(* Logix 5000 project; controller cal1632 1756-L62 rev 16.20; software revision 16.05; part 19 of 61 *)
(* tags used below, declared in another part *)
   FAULT : BOOL;
   p01_param_fan_zero_speed : REAL;
   p01_param_open_oven_recirc_sp : REAL;
   p01_param_temp_limit : REAL;
   p01_recipe_active : recipe;
   p01r02 : routine;
   p01r09_open_oven : BOOL;
   p01r09_pb_global_reset : BOOL;
   p02_dint_from_hmi : hmi_dint;
   p11r02_shutdown_temp : BOOL;
   p11r30 : routine;
   p12_ai_recirc_rpm : REAL;
   p12_ao_recirc_selected_speed : REAL;
   p12_di_recirc : acs800_di_normal;
   p12_di_recirc_fan_mtr_ts : BOOL;
   p12_di_recirc_flow_ok : BOOL;
   p12_do_recirc : acs800_do_normal;
   p12r02_shutdown_temp : BOOL;
   p12r20_state : DINT;
   p12r30 : routine;
   p12r32 : routine;
   p12r32_fan_pb_stopped : BOOL;
   p12r32_pb_start : BOOL;
   p12r32_pb_stop : BOOL;
   p12r32_request_auto_run : BOOL;
   p12r32_run_permissive : BOOL;
   p12r32_timer_fault : TIMER[5];
   p12r32_timer_warning : TIMER[5];
   p12r32_vfd_stopped : BOOL;
   p13_ai_exhaust_amps : REAL;
   p13_ai_exhaust_hz : REAL;
   p13_ai_exhaust_hz_max : REAL;
   p13_ai_exhaust_rpm : REAL;
   p13_ai_recirc_amps : REAL;
   p13_ai_recirc_hz : REAL;
   p13_ai_recirc_hz_max : REAL;
   p13_ai_recirc_rpm : REAL;
   p13_ai_tc01 : REAL;
   p13_ai_tc02 : REAL;
   p13_di_door_open : BOOL;
   p13_di_exh : acs800_di_normal;
   p13_di_exh_fan_mtr_ts : BOOL;
   p13_di_exh_flow_ok : BOOL;
   p13_di_filter_clean : BOOL;
   p13_di_recirc : acs800_di_normal;
   p13_di_recirc_fan_mtr_ts : BOOL;
   p13_di_recirc_flow_ok : BOOL;
   p13_di_tc01_bo : BOOL;
   p13_di_tc02_bo : BOOL;
   p13_dint_to_hmi : DINT[16];
   p13_param_shutdown_temp : REAL;
   p13_param_tc01z : REAL;
   p13_param_tc02z : REAL;
   p13r01 : routine;
   p13r02 : routine;
   p13r02_fault_exists : BOOL;
   p13r02_not_safe_temp : BOOL;
   p13r02_safe_temp : BOOL;
   p13r02_shutdown_temp : BOOL;
   p13r02_timer_fault : TIMER[4];
   p13r02_timer_safe_temp : TIMER[2];
   p13r02_timer_warning : TIMER[4];
   p13r02_unack_fault : BOOL;
   p13r02_unack_warning : BOOL;
   p13r02_warning_exists : BOOL;
   p13r03 : routine;
   p13r03_hz : SYS_SCP;
   p13r03_timer_fault : TIMER[4];
   p13r03_timer_warning : TIMER[4];
   p13r04 : routine;
   p13r05 : routine;
   p13r06 : routine;
   p13r07 : routine;
   p13r08 : routine;
   p13r09 : routine;
   p13r10 : routine;
   p13r20 : routine;
   p13r30 : routine;
   p13r31 : routine;
   p13r32 : routine;
   p23r02 : routine;
(* P12_Zone_2, continued *)

ROUTINE R32_Recirc_VFD   (* ladder *)
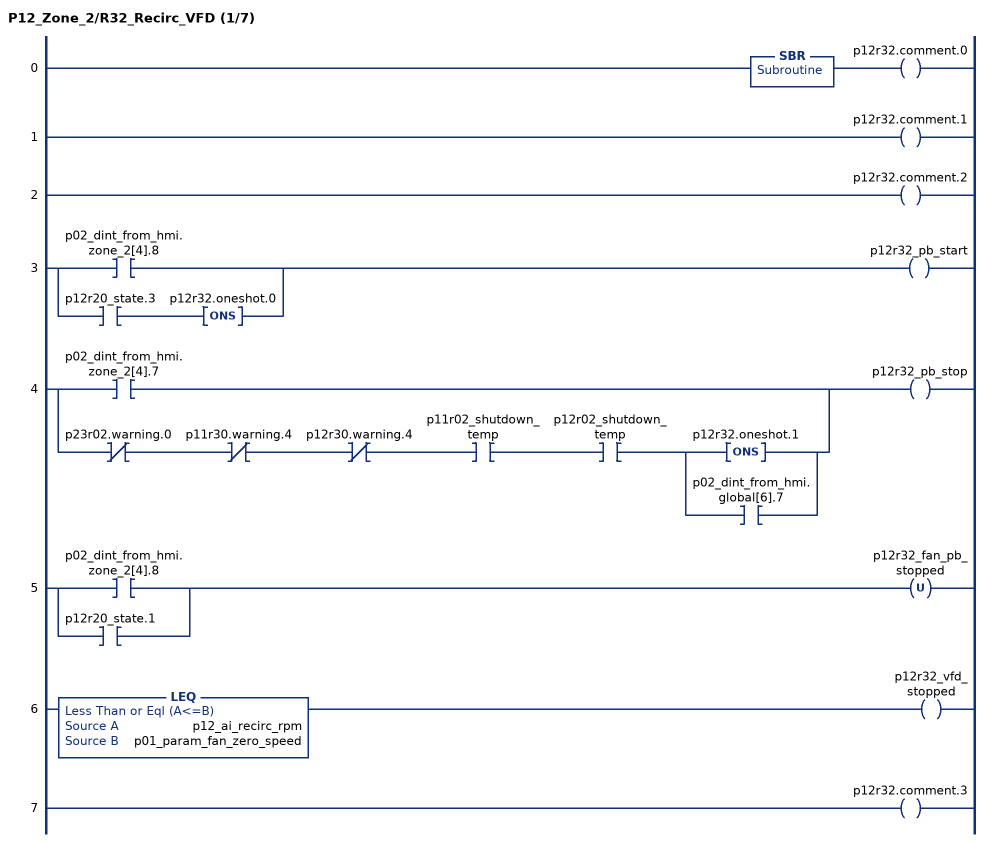
   0: SBR()OTE(p12r32.comment.0);
   1: OTE(p12r32.comment.1);
   2: OTE(p12r32.comment.2);
   3: [XIC(p02_dint_from_hmi.zone_2[4].8) ,XIC(p12r20_state.3) ONS(p12r32.oneshot.0) ]OTE(p12r32_pb_start);
   4: [XIC(p02_dint_from_hmi.zone_2[4].7) ,XIO(p23r02.warning.0) XIO(p11r30.warning.4) XIO(p12r30.warning.4) XIC(p11r02_shutdown_temp) XIC(p12r02_shutdown_temp) [ONS(p12r32.oneshot.1) ,XIC(p02_dint_from_hmi.global[6].7) ] ]OTE(p12r32_pb_stop);
   5: [XIC(p02_dint_from_hmi.zone_2[4].8) ,XIC(p12r20_state.1) ]OTU(p12r32_fan_pb_stopped);
   6: LEQ(p12_ai_recirc_rpm,p01_param_fan_zero_speed)OTE(p12r32_vfd_stopped);
   7: OTE(p12r32.comment.3);
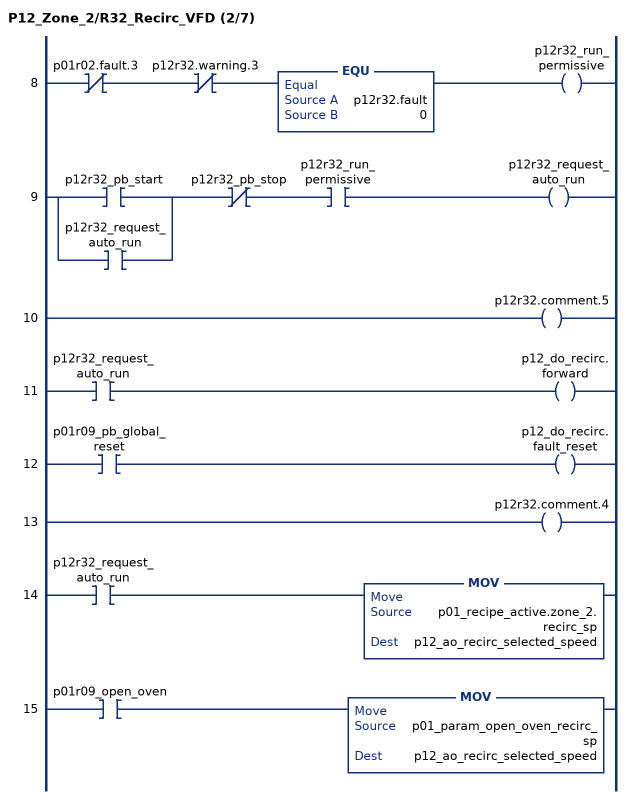
   8: XIO(p01r02.fault.3)XIO(p12r32.warning.3)EQU(p12r32.fault,0)OTE(p12r32_run_permissive);
   9: [XIC(p12r32_pb_start) ,XIC(p12r32_request_auto_run) ]XIO(p12r32_pb_stop)XIC(p12r32_run_permissive)OTE(p12r32_request_auto_run);
   10: OTE(p12r32.comment.5);
   11: XIC(p12r32_request_auto_run)OTE(p12_do_recirc.forward);
   12: XIC(p01r09_pb_global_reset)OTE(p12_do_recirc.fault_reset);
   13: OTE(p12r32.comment.4);
   14: XIC(p12r32_request_auto_run)MOV(p01_recipe_active.zone_2.recirc_sp,p12_ao_recirc_selected_speed);
   15: XIC(p01r09_open_oven)MOV(p01_param_open_oven_recirc_sp,p12_ao_recirc_selected_speed);
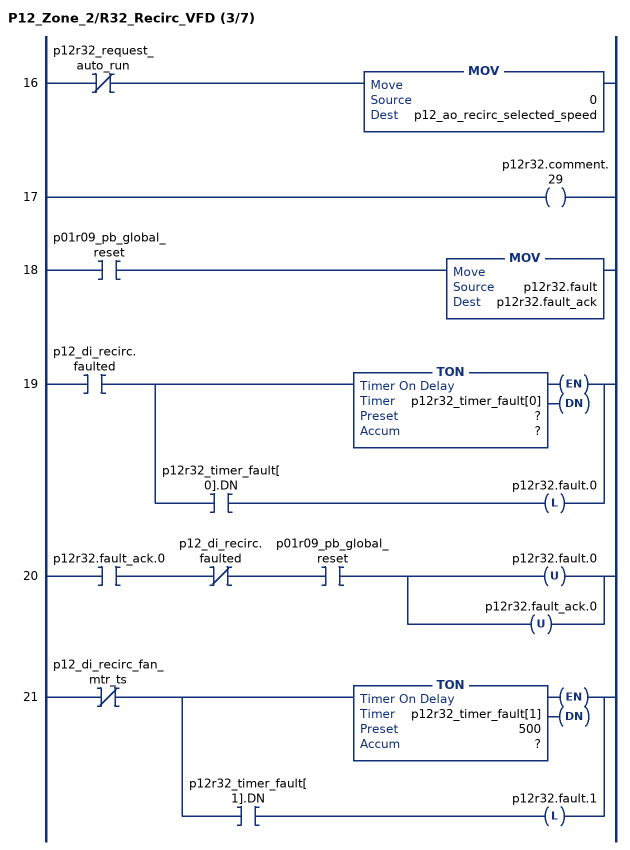
   16: XIO(p12r32_request_auto_run)MOV(0,p12_ao_recirc_selected_speed);
   17: OTE(p12r32.comment.29);
   18: XIC(p01r09_pb_global_reset)MOV(p12r32.fault,p12r32.fault_ack);
   19: XIC(p12_di_recirc.faulted)[TON(p12r32_timer_fault[0],?,?) ,XIC(p12r32_timer_fault[0].DN) OTL(p12r32.fault.0) ];
   20: XIC(p12r32.fault_ack.0)XIO(p12_di_recirc.faulted)XIC(p01r09_pb_global_reset)[OTU(p12r32.fault.0) ,OTU(p12r32.fault_ack.0) ];
   21: XIO(p12_di_recirc_fan_mtr_ts)[TON(p12r32_timer_fault[1],?,?) ,XIC(p12r32_timer_fault[1].DN) OTL(p12r32.fault.1) ];
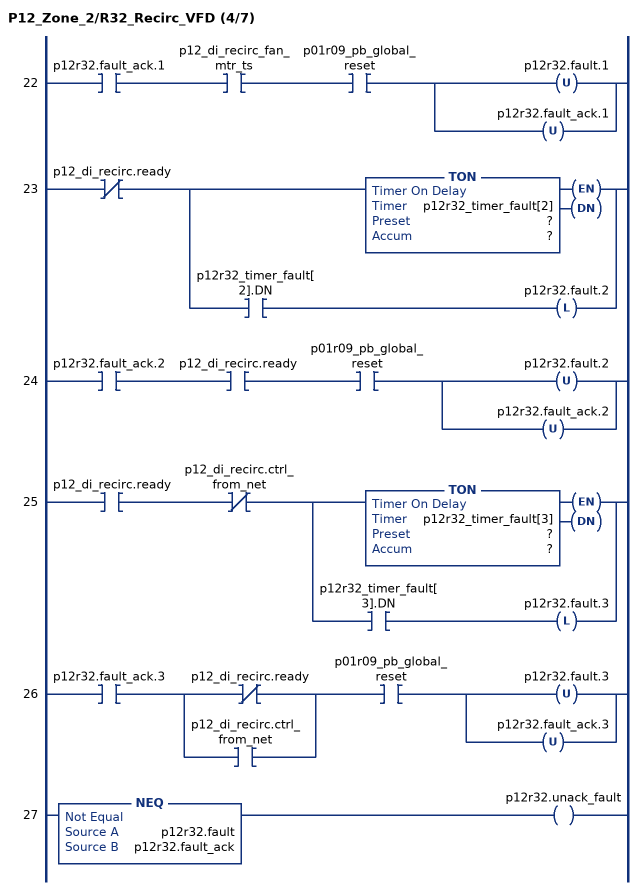
   22: XIC(p12r32.fault_ack.1)XIC(p12_di_recirc_fan_mtr_ts)XIC(p01r09_pb_global_reset)[OTU(p12r32.fault.1) ,OTU(p12r32.fault_ack.1) ];
   23: XIO(p12_di_recirc.ready)[TON(p12r32_timer_fault[2],?,?) ,XIC(p12r32_timer_fault[2].DN) OTL(p12r32.fault.2) ];
   24: XIC(p12r32.fault_ack.2)XIC(p12_di_recirc.ready)XIC(p01r09_pb_global_reset)[OTU(p12r32.fault.2) ,OTU(p12r32.fault_ack.2) ];
   25: XIC(p12_di_recirc.ready)XIO(p12_di_recirc.ctrl_from_net)[TON(p12r32_timer_fault[3],?,?) ,XIC(p12r32_timer_fault[3].DN) OTL(p12r32.fault.3) ];
   26: XIC(p12r32.fault_ack.3)[XIO(p12_di_recirc.ready) ,XIC(p12_di_recirc.ctrl_from_net) ]XIC(p01r09_pb_global_reset)[OTU(p12r32.fault.3) ,OTU(p12r32.fault_ack.3) ];
   27: NEQ(p12r32.fault,p12r32.fault_ack)OTE(p12r32.unack_fault);
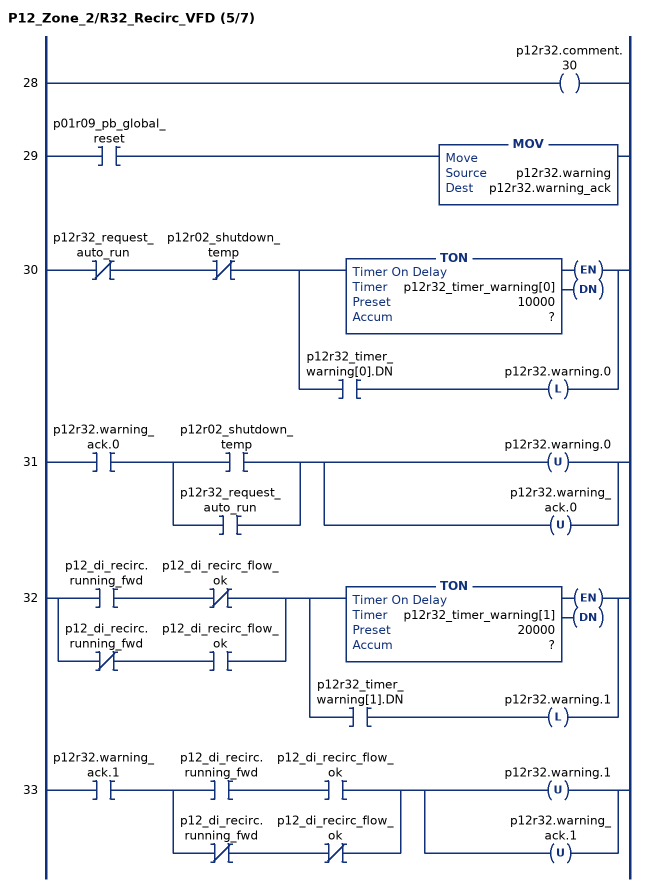
   28: OTE(p12r32.comment.30);
   29: XIC(p01r09_pb_global_reset)MOV(p12r32.warning,p12r32.warning_ack);
   30: XIO(p12r32_request_auto_run)XIO(p12r02_shutdown_temp)[TON(p12r32_timer_warning[0],?,?) ,XIC(p12r32_timer_warning[0].DN) OTL(p12r32.warning.0) ];
   31: XIC(p12r32.warning_ack.0)[XIC(p12r02_shutdown_temp) ,XIC(p12r32_request_auto_run) ][OTU(p12r32.warning.0) ,OTU(p12r32.warning_ack.0) ];
   32: [XIC(p12_di_recirc.running_fwd) XIO(p12_di_recirc_flow_ok) ,XIO(p12_di_recirc.running_fwd) XIC(p12_di_recirc_flow_ok) ][TON(p12r32_timer_warning[1],?,?) ,XIC(p12r32_timer_warning[1].DN) OTL(p12r32.warning.1) ];
   33: XIC(p12r32.warning_ack.1)[XIC(p12_di_recirc.running_fwd) XIC(p12_di_recirc_flow_ok) ,XIO(p12_di_recirc.running_fwd) XIO(p12_di_recirc_flow_ok) ][OTU(p12r32.warning.1) ,OTU(p12r32.warning_ack.1) ];
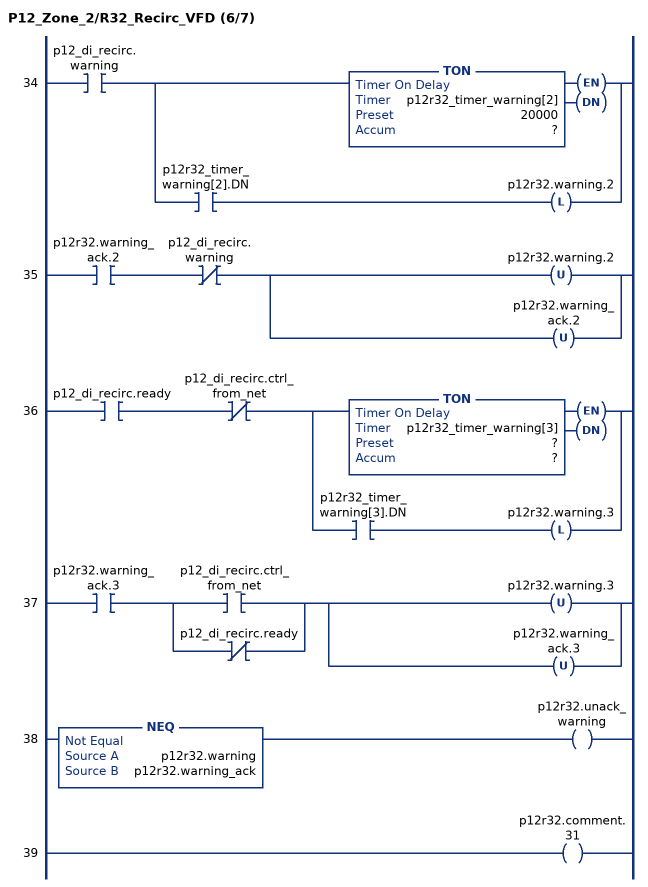
   34: XIC(p12_di_recirc.warning)[TON(p12r32_timer_warning[2],?,?) ,XIC(p12r32_timer_warning[2].DN) OTL(p12r32.warning.2) ];
   35: XIC(p12r32.warning_ack.2)XIO(p12_di_recirc.warning)[OTU(p12r32.warning.2) ,OTU(p12r32.warning_ack.2) ];
   36: XIC(p12_di_recirc.ready)XIO(p12_di_recirc.ctrl_from_net)[TON(p12r32_timer_warning[3],?,?) ,XIC(p12r32_timer_warning[3].DN) OTL(p12r32.warning.3) ];
   37: XIC(p12r32.warning_ack.3)[XIC(p12_di_recirc.ctrl_from_net) ,XIO(p12_di_recirc.ready) ][OTU(p12r32.warning.3) ,OTU(p12r32.warning_ack.3) ];
   38: NEQ(p12r32.warning,p12r32.warning_ack)OTE(p12r32.unack_warning);
   39: OTE(p12r32.comment.31);
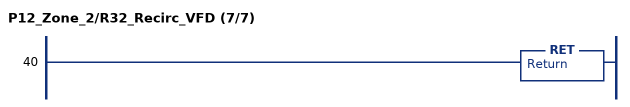
   40: RET();
END_ROUTINE
END_PROGRAM

PROGRAM P13_Zone_3   (* main routine R01_Main *)

ROUTINE R01_Main   (* ladder *)
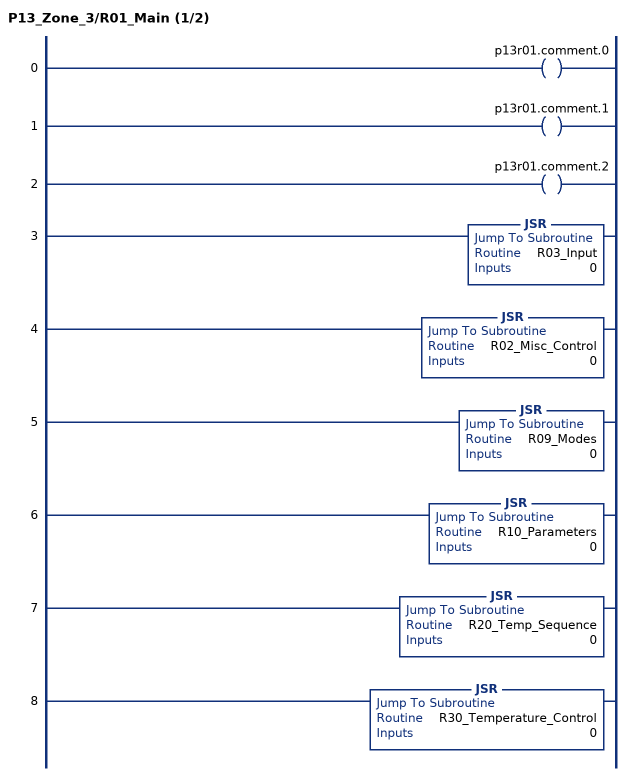
   0: OTE(p13r01.comment.0);
   1: OTE(p13r01.comment.1);
   2: OTE(p13r01.comment.2);
   3: JSR(R03_Input,0);
   4: JSR(R02_Misc_Control,0);
   5: JSR(R09_Modes,0);
   6: JSR(R10_Parameters,0);
   7: JSR(R20_Temp_Sequence,0);
   8: JSR(R30_Temperature_Control,0);
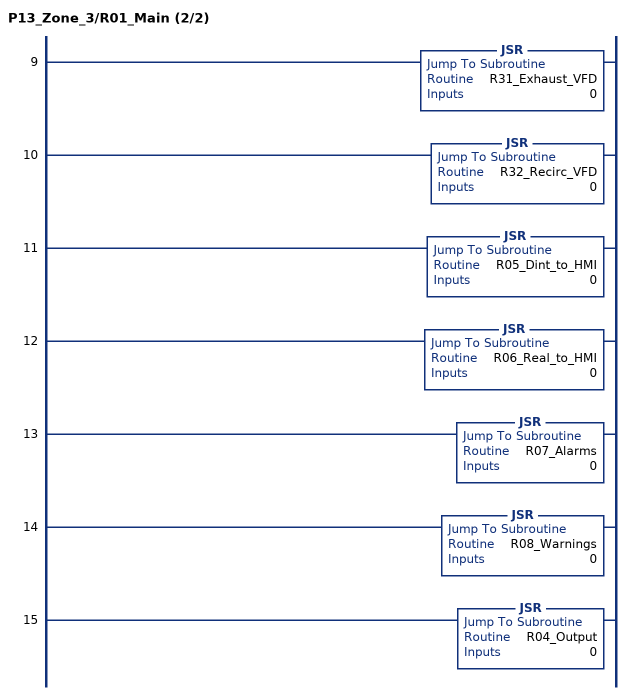
   9: JSR(R31_Exhaust_VFD,0);
   10: JSR(R32_Recirc_VFD,0);
   11: JSR(R05_Dint_to_HMI,0);
   12: JSR(R06_Real_to_HMI,0);
   13: JSR(R07_Alarms,0);
   14: JSR(R08_Warnings,0);
   15: JSR(R04_Output,0);
END_ROUTINE

ROUTINE R02_Misc_Control   (* ladder *)
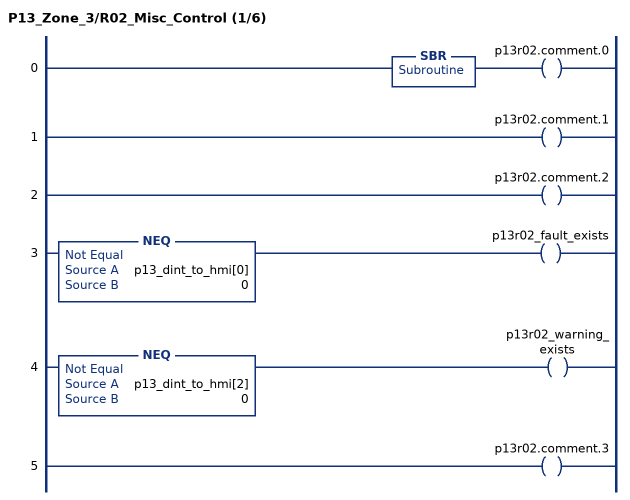
   0: SBR()OTE(p13r02.comment.0);
   1: OTE(p13r02.comment.1);
   2: OTE(p13r02.comment.2);
   3: NEQ(p13_dint_to_hmi[0],0)OTE(p13r02_fault_exists);
   4: NEQ(p13_dint_to_hmi[2],0)OTE(p13r02_warning_exists);
   5: OTE(p13r02.comment.3);
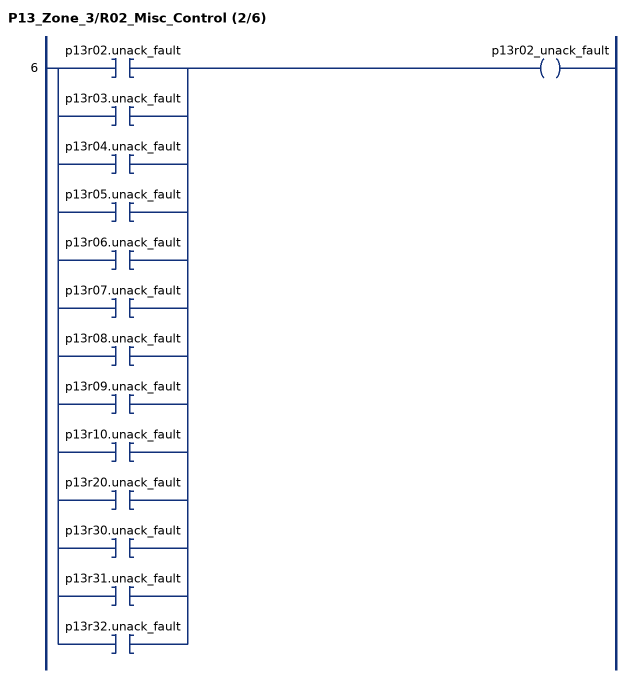
   6: [XIC(p13r02.unack_fault) ,XIC(p13r03.unack_fault) ,XIC(p13r04.unack_fault) ,XIC(p13r05.unack_fault) ,XIC(p13r06.unack_fault) ,XIC(p13r07.unack_fault) ,XIC(p13r08.unack_fault) ,XIC(p13r09.unack_fault) ,XIC(p13r10.unack_fault) ,XIC(p13r20.unack_fault) ,XIC(p13r30.unack_fault) ,XIC(p13r31.unack_fault) ,XIC(p13r32.unack_fault) ]OTE(p13r02_unack_fault);
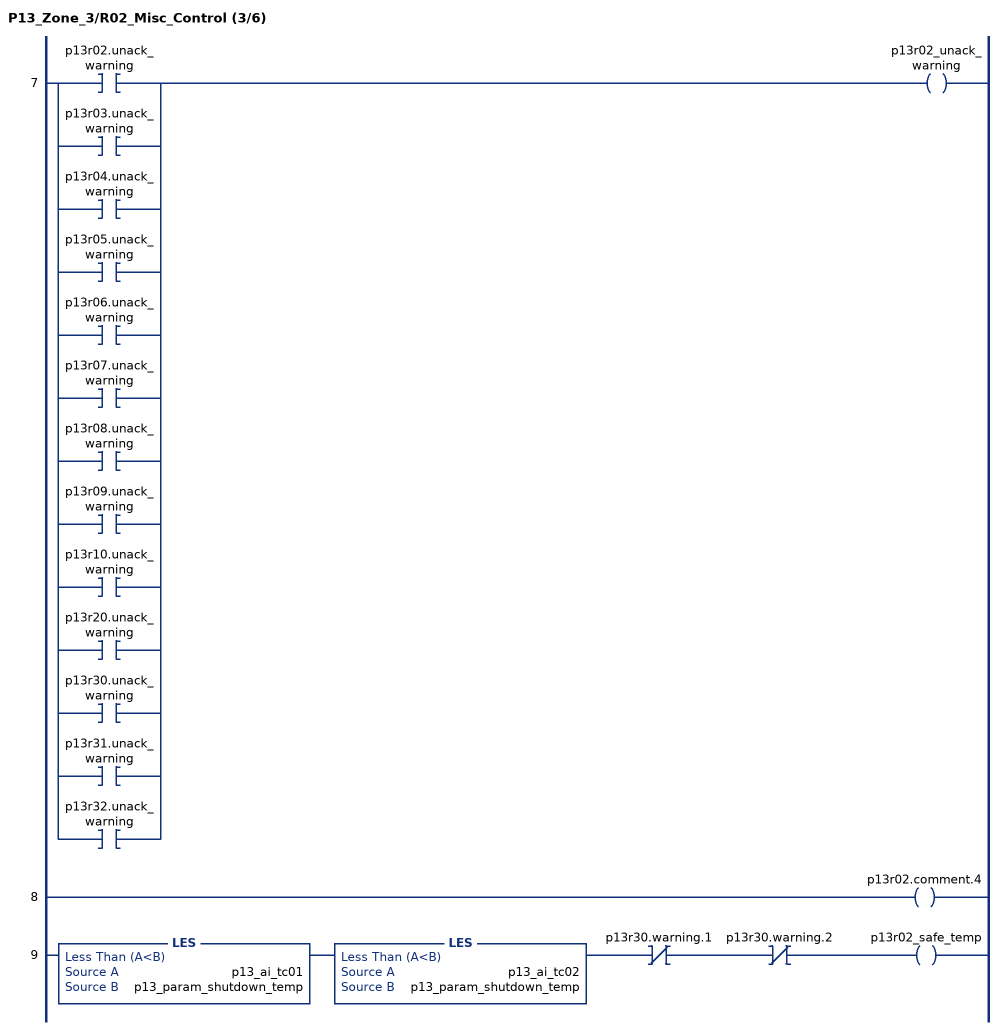
   7: [XIC(p13r02.unack_warning) ,XIC(p13r03.unack_warning) ,XIC(p13r04.unack_warning) ,XIC(p13r05.unack_warning) ,XIC(p13r06.unack_warning) ,XIC(p13r07.unack_warning) ,XIC(p13r08.unack_warning) ,XIC(p13r09.unack_warning) ,XIC(p13r10.unack_warning) ,XIC(p13r20.unack_warning) ,XIC(p13r30.unack_warning) ,XIC(p13r31.unack_warning) ,XIC(p13r32.unack_warning) ]OTE(p13r02_unack_warning);
   8: OTE(p13r02.comment.4);
   9: LES(p13_ai_tc01,p13_param_shutdown_temp)LES(p13_ai_tc02,p13_param_shutdown_temp)XIO(p13r30.warning.1)XIO(p13r30.warning.2)OTE(p13r02_safe_temp);
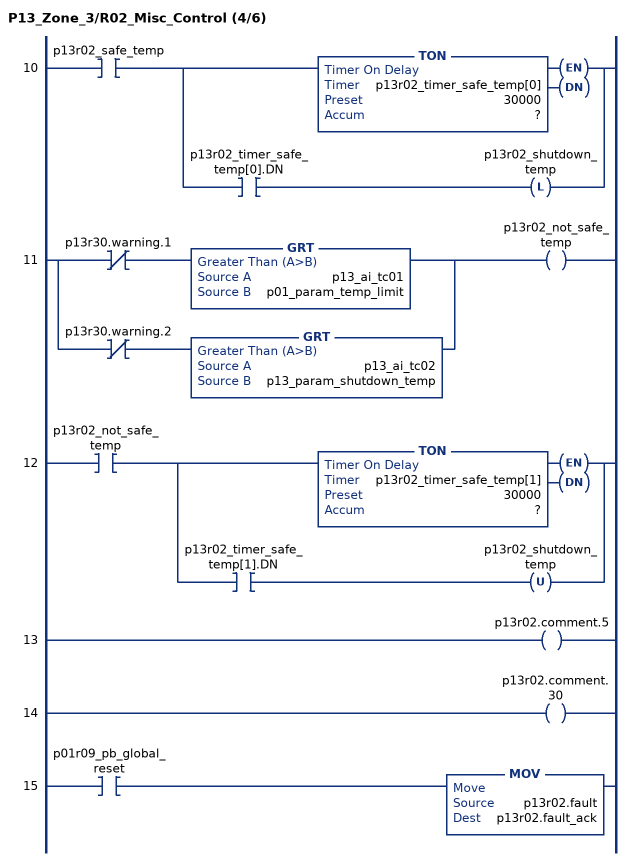
   10: XIC(p13r02_safe_temp)[TON(p13r02_timer_safe_temp[0],?,?) ,XIC(p13r02_timer_safe_temp[0].DN) OTL(p13r02_shutdown_temp) ];
   11: [XIO(p13r30.warning.1) GRT(p13_ai_tc01,p01_param_temp_limit) ,XIO(p13r30.warning.2) GRT(p13_ai_tc02,p13_param_shutdown_temp) ]OTE(p13r02_not_safe_temp);
   12: XIC(p13r02_not_safe_temp)[TON(p13r02_timer_safe_temp[1],?,?) ,XIC(p13r02_timer_safe_temp[1].DN) OTU(p13r02_shutdown_temp) ];
   13: OTE(p13r02.comment.5);
   14: OTE(p13r02.comment.30);
   15: XIC(p01r09_pb_global_reset)MOV(p13r02.fault,p13r02.fault_ack);
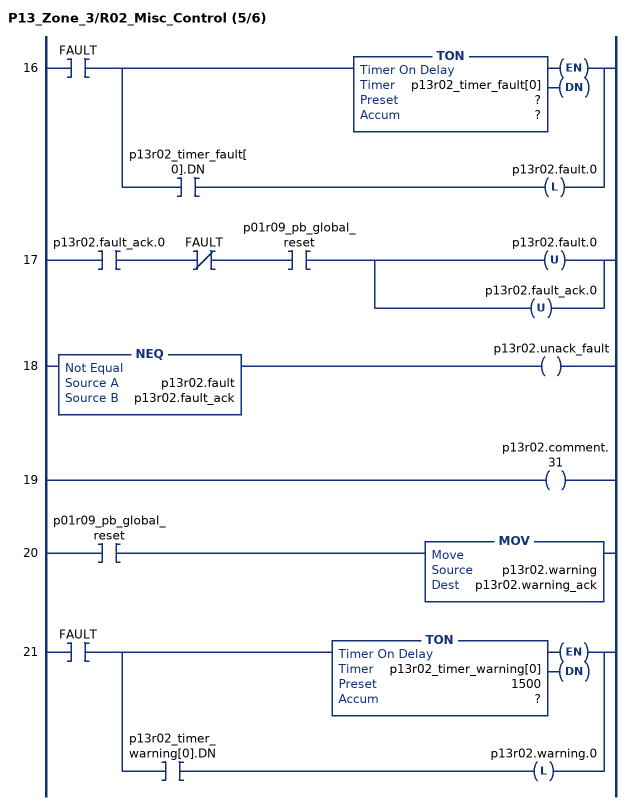
   16: XIC(FAULT)[TON(p13r02_timer_fault[0],?,?) ,XIC(p13r02_timer_fault[0].DN) OTL(p13r02.fault.0) ];
   17: XIC(p13r02.fault_ack.0)XIO(FAULT)XIC(p01r09_pb_global_reset)[OTU(p13r02.fault.0) ,OTU(p13r02.fault_ack.0) ];
   18: NEQ(p13r02.fault,p13r02.fault_ack)OTE(p13r02.unack_fault);
   19: OTE(p13r02.comment.31);
   20: XIC(p01r09_pb_global_reset)MOV(p13r02.warning,p13r02.warning_ack);
   21: XIC(FAULT)[TON(p13r02_timer_warning[0],?,?) ,XIC(p13r02_timer_warning[0].DN) OTL(p13r02.warning.0) ];
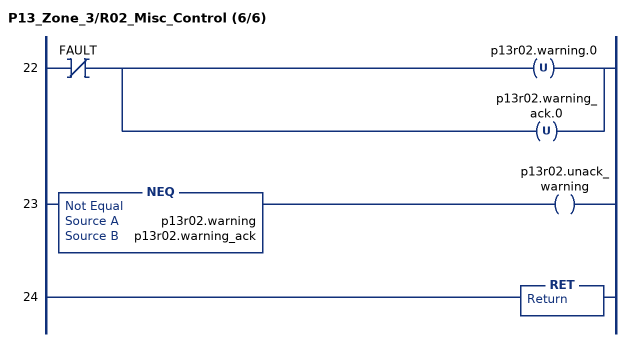
   22: XIO(FAULT)[OTU(p13r02.warning.0) ,OTU(p13r02.warning_ack.0) ];
   23: NEQ(p13r02.warning,p13r02.warning_ack)OTE(p13r02.unack_warning);
   24: RET();
END_ROUTINE

ROUTINE R03_Input   (* ladder *)
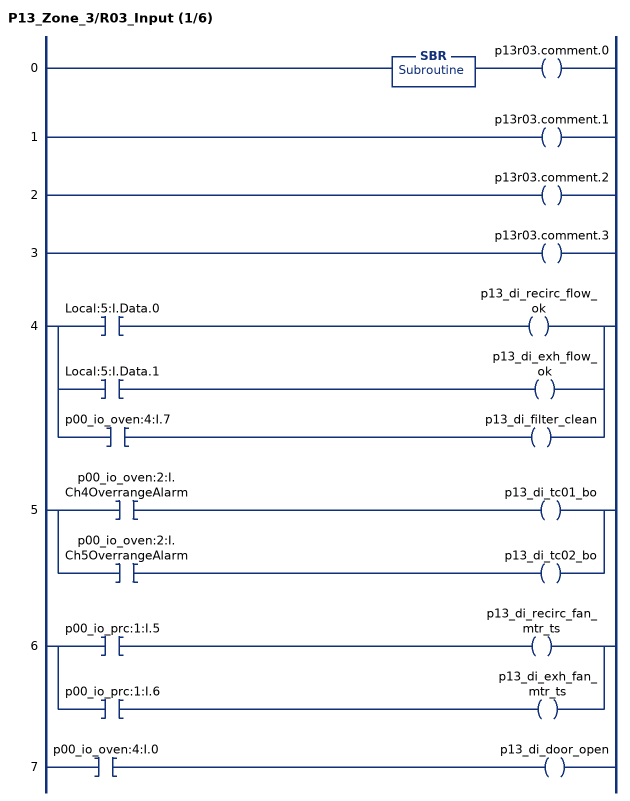
   0: SBR()OTE(p13r03.comment.0);
   1: OTE(p13r03.comment.1);
   2: OTE(p13r03.comment.2);
   3: OTE(p13r03.comment.3);
   4: [XIC(Local:5:I.Data.0) OTE(p13_di_recirc_flow_ok) ,XIC(Local:5:I.Data.1) OTE(p13_di_exh_flow_ok) ,XIC(p00_io_oven:4:I.7) OTE(p13_di_filter_clean) ];
   5: [XIC(p00_io_oven:2:I.Ch4OverrangeAlarm) OTE(p13_di_tc01_bo) ,XIC(p00_io_oven:2:I.Ch5OverrangeAlarm) OTE(p13_di_tc02_bo) ];
   6: [XIC(p00_io_prc:1:I.5) OTE(p13_di_recirc_fan_mtr_ts) ,XIC(p00_io_prc:1:I.6) OTE(p13_di_exh_fan_mtr_ts) ];
   7: XIC(p00_io_oven:4:I.0)OTE(p13_di_door_open);
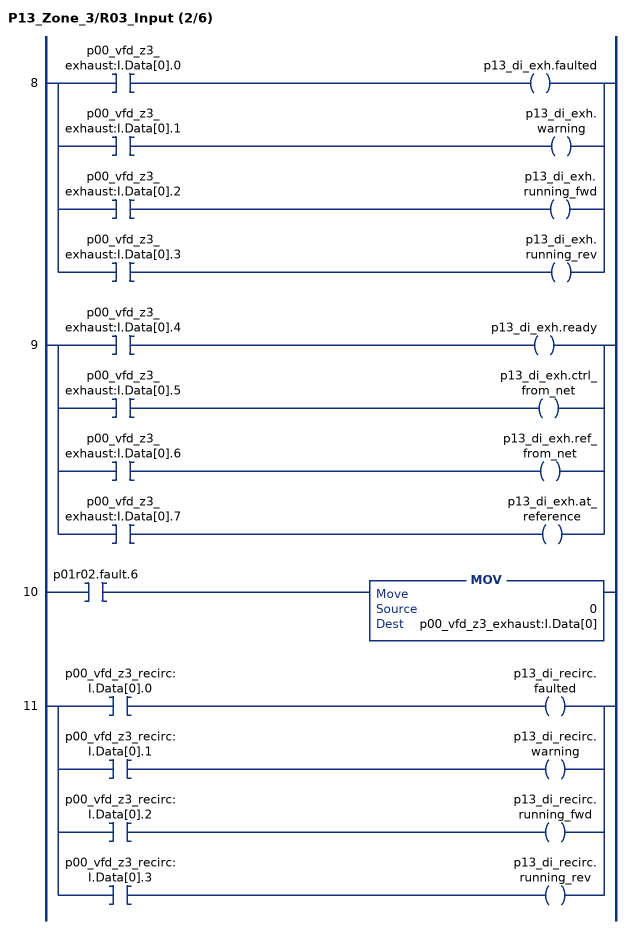
   8: [XIC(p00_vfd_z3_exhaust:I.Data[0].0) OTE(p13_di_exh.faulted) ,XIC(p00_vfd_z3_exhaust:I.Data[0].1) OTE(p13_di_exh.warning) ,XIC(p00_vfd_z3_exhaust:I.Data[0].2) OTE(p13_di_exh.running_fwd) ,XIC(p00_vfd_z3_exhaust:I.Data[0].3) OTE(p13_di_exh.running_rev) ];
   9: [XIC(p00_vfd_z3_exhaust:I.Data[0].4) OTE(p13_di_exh.ready) ,XIC(p00_vfd_z3_exhaust:I.Data[0].5) OTE(p13_di_exh.ctrl_from_net) ,XIC(p00_vfd_z3_exhaust:I.Data[0].6) OTE(p13_di_exh.ref_from_net) ,XIC(p00_vfd_z3_exhaust:I.Data[0].7) OTE(p13_di_exh.at_reference) ];
   10: XIC(p01r02.fault.6)MOV(0,p00_vfd_z3_exhaust:I.Data[0]);
   11: [XIC(p00_vfd_z3_recirc:I.Data[0].0) OTE(p13_di_recirc.faulted) ,XIC(p00_vfd_z3_recirc:I.Data[0].1) OTE(p13_di_recirc.warning) ,XIC(p00_vfd_z3_recirc:I.Data[0].2) OTE(p13_di_recirc.running_fwd) ,XIC(p00_vfd_z3_recirc:I.Data[0].3) OTE(p13_di_recirc.running_rev) ];
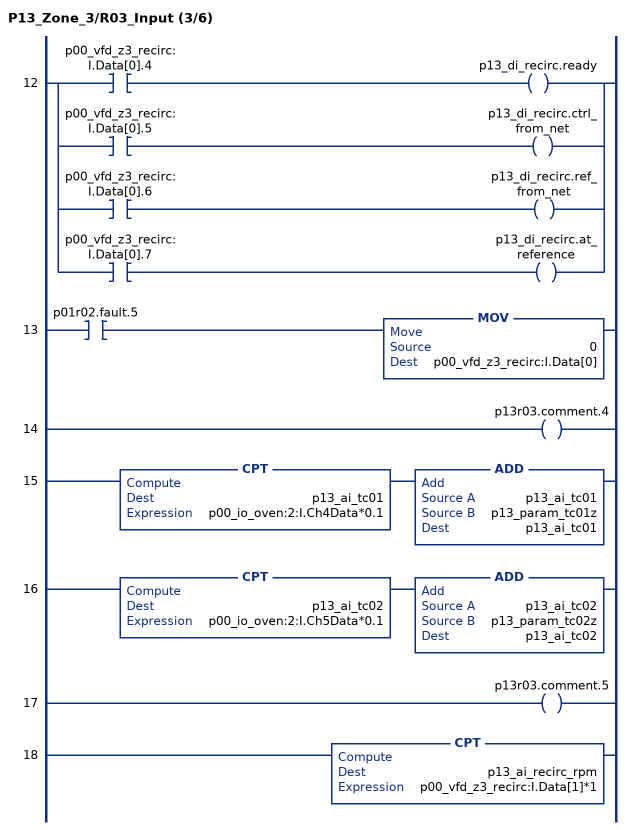
   12: [XIC(p00_vfd_z3_recirc:I.Data[0].4) OTE(p13_di_recirc.ready) ,XIC(p00_vfd_z3_recirc:I.Data[0].5) OTE(p13_di_recirc.ctrl_from_net) ,XIC(p00_vfd_z3_recirc:I.Data[0].6) OTE(p13_di_recirc.ref_from_net) ,XIC(p00_vfd_z3_recirc:I.Data[0].7) OTE(p13_di_recirc.at_reference) ];
   13: XIC(p01r02.fault.5)MOV(0,p00_vfd_z3_recirc:I.Data[0]);
   14: OTE(p13r03.comment.4);
   15: CPT(p13_ai_tc01,p00_io_oven:2:I.Ch4Data*0.1)ADD(p13_ai_tc01,p13_param_tc01z,p13_ai_tc01);
   16: CPT(p13_ai_tc02,p00_io_oven:2:I.Ch5Data*0.1)ADD(p13_ai_tc02,p13_param_tc02z,p13_ai_tc02);
   17: OTE(p13r03.comment.5);
   18: CPT(p13_ai_recirc_rpm,p00_vfd_z3_recirc:I.Data[1]*1);
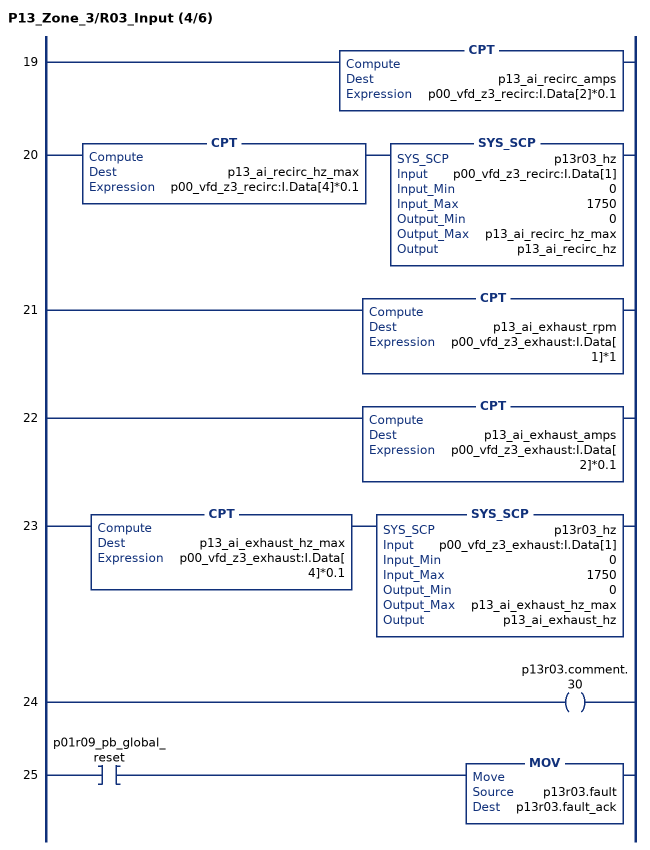
   19: CPT(p13_ai_recirc_amps,p00_vfd_z3_recirc:I.Data[2]*0.1);
   20: CPT(p13_ai_recirc_hz_max,p00_vfd_z3_recirc:I.Data[4]*0.1)SYS_SCP(p13r03_hz,p00_vfd_z3_recirc:I.Data[1],0,1750,0,p13_ai_recirc_hz_max,p13_ai_recirc_hz);
   21: CPT(p13_ai_exhaust_rpm,p00_vfd_z3_exhaust:I.Data[1]*1);
   22: CPT(p13_ai_exhaust_amps,p00_vfd_z3_exhaust:I.Data[2]*0.1);
   23: CPT(p13_ai_exhaust_hz_max,p00_vfd_z3_exhaust:I.Data[4]*0.1)SYS_SCP(p13r03_hz,p00_vfd_z3_exhaust:I.Data[1],0,1750,0,p13_ai_exhaust_hz_max,p13_ai_exhaust_hz);
   24: OTE(p13r03.comment.30);
   25: XIC(p01r09_pb_global_reset)MOV(p13r03.fault,p13r03.fault_ack);
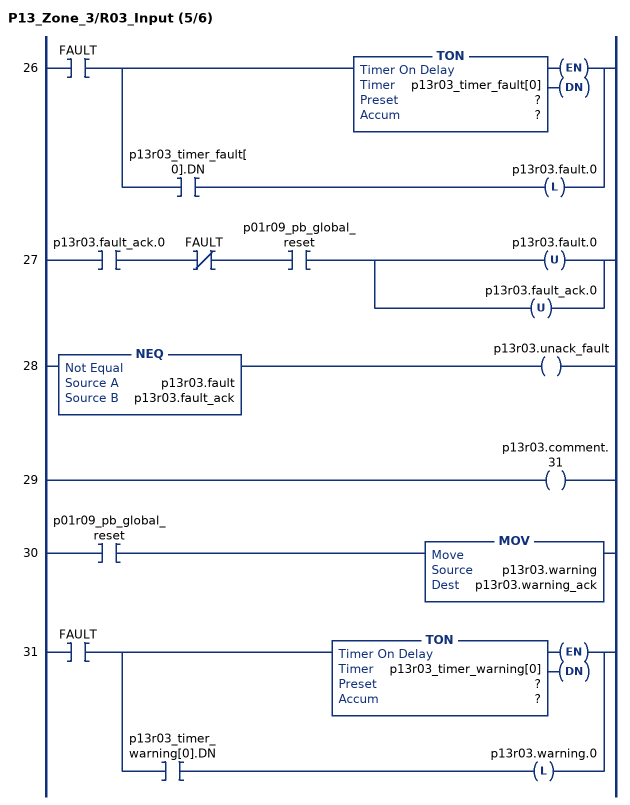
   26: XIC(FAULT)[TON(p13r03_timer_fault[0],?,?) ,XIC(p13r03_timer_fault[0].DN) OTL(p13r03.fault.0) ];
   27: XIC(p13r03.fault_ack.0)XIO(FAULT)XIC(p01r09_pb_global_reset)[OTU(p13r03.fault.0) ,OTU(p13r03.fault_ack.0) ];
   28: NEQ(p13r03.fault,p13r03.fault_ack)OTE(p13r03.unack_fault);
   29: OTE(p13r03.comment.31);
   30: XIC(p01r09_pb_global_reset)MOV(p13r03.warning,p13r03.warning_ack);
   31: XIC(FAULT)[TON(p13r03_timer_warning[0],?,?) ,XIC(p13r03_timer_warning[0].DN) OTL(p13r03.warning.0) ];
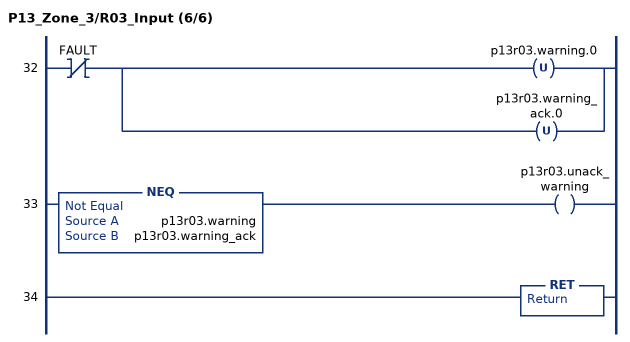
   32: XIO(FAULT)[OTU(p13r03.warning.0) ,OTU(p13r03.warning_ack.0) ];
   33: NEQ(p13r03.warning,p13r03.warning_ack)OTE(p13r03.unack_warning);
   34: RET();
END_ROUTINE
